// TIA Portal V17 export
// export: Created 2021-09-01T12:00:00, ExportSetting None, DisplayName Totally Integrated Automation Portal, DisplayVersion V17 Update 6
FUNCTION_BLOCK "DEMOSCHRITTKETTE"   // FB45, LAD
TITLE = DemoSchrittKette
{ S7_Optimized_Access := 'TRUE' }
// Auto genereted sequence by graph2LAD: 2024-11-19
// E.R. https://github.com/eliasrhoden
// stored: MemoryReserve 100, SetENOAutomatically false
   VAR_INPUT
      enable : Bool;   // Enables the state machine
      reset : Bool;   // Resets to init state
   END_VAR
   VAR
      statStep : Int;   // Current step/state
      statNextStep : Int;   // Step/State next PLC cycle
   END_VAR
   VAR CONSTANT
      INIT : Int := 0;
      GOTO_HOME : Int := 10;
      AT_HOME_POS : Int := 20;
      LOADING : Int := 30;
      WORKING : Int := 40;
      UNLOADING : Int := 50;
   END_VAR
   VAR_TEMP   // added for the SCL form of the ladder/FBD networks
      _w1 : Bool;
   END_VAR
BEGIN

REGION Network 1 (SCL): Reset
   IF #reset THEN
    #statStep := #INIT;
    #statNextStep := #INIT;
   END_IF;
END_REGION

REGION Network 2: INIT
   // INIT
   // 	 -> GOTO_HOME 
   // 	 -> UNLOADING
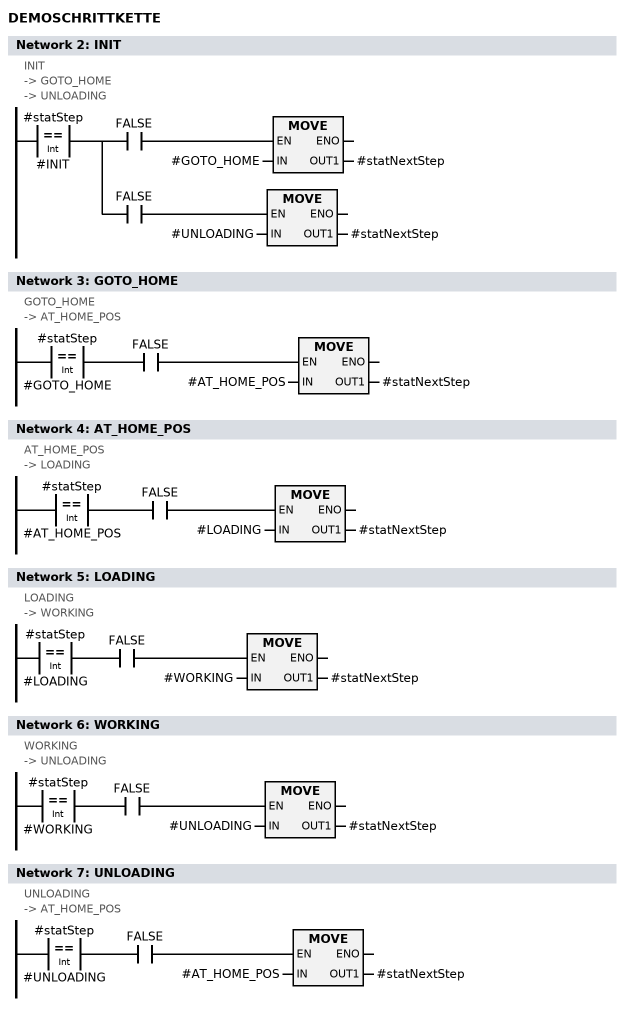
   RUNG wire#powerrail
      { S7_Templates := "SrcType := Int" } EQ_Contact(in1 := #statStep, in2 := #INIT)
      wire#w1
      Contact( FALSE )
      Move(in := #GOTO_HOME, out1 => #statNextStep)
   END_RUNG
   RUNG wire#w1
      Contact( FALSE )
      Move(in := #UNLOADING, out1 => #statNextStep)
   END_RUNG
   // the same network as SCL:
   #_w1 := #statStep = #INIT;
   IF #_w1 AND FALSE THEN
       #statNextStep := #GOTO_HOME;
       #statNextStep := #UNLOADING;
   END_IF;
END_REGION

REGION Network 3: GOTO_HOME
   // GOTO_HOME
   // 	 -> AT_HOME_POS
   RUNG wire#powerrail
      { S7_Templates := "SrcType := Int" } EQ_Contact(in1 := #statStep, in2 := #GOTO_HOME)
      Contact( FALSE )
      Move(in := #AT_HOME_POS, out1 => #statNextStep)
   END_RUNG
   // the same network as SCL:
   IF (#statStep = #GOTO_HOME) AND FALSE THEN #statNextStep := #AT_HOME_POS; END_IF;
END_REGION

REGION Network 4: AT_HOME_POS
   // AT_HOME_POS
   // 	 -> LOADING
   RUNG wire#powerrail
      { S7_Templates := "SrcType := Int" } EQ_Contact(in1 := #statStep, in2 := #AT_HOME_POS)
      Contact( FALSE )
      Move(in := #LOADING, out1 => #statNextStep)
   END_RUNG
   // the same network as SCL:
   IF (#statStep = #AT_HOME_POS) AND FALSE THEN #statNextStep := #LOADING; END_IF;
END_REGION

REGION Network 5: LOADING
   // LOADING
   // 	 -> WORKING
   RUNG wire#powerrail
      { S7_Templates := "SrcType := Int" } EQ_Contact(in1 := #statStep, in2 := #LOADING)
      Contact( FALSE )
      Move(in := #WORKING, out1 => #statNextStep)
   END_RUNG
   // the same network as SCL:
   IF (#statStep = #LOADING) AND FALSE THEN #statNextStep := #WORKING; END_IF;
END_REGION

REGION Network 6: WORKING
   // WORKING
   // 	 -> UNLOADING
   RUNG wire#powerrail
      { S7_Templates := "SrcType := Int" } EQ_Contact(in1 := #statStep, in2 := #WORKING)
      Contact( FALSE )
      Move(in := #UNLOADING, out1 => #statNextStep)
   END_RUNG
   // the same network as SCL:
   IF (#statStep = #WORKING) AND FALSE THEN #statNextStep := #UNLOADING; END_IF;
END_REGION

REGION Network 7: UNLOADING
   // UNLOADING
   // 	 -> AT_HOME_POS
   RUNG wire#powerrail
      { S7_Templates := "SrcType := Int" } EQ_Contact(in1 := #statStep, in2 := #UNLOADING)
      Contact( FALSE )
      Move(in := #AT_HOME_POS, out1 => #statNextStep)
   END_RUNG
   // the same network as SCL:
   IF (#statStep = #UNLOADING) AND FALSE THEN #statNextStep := #AT_HOME_POS; END_IF;
END_REGION

REGION Network 8 (SCL): Next step
   // This ensurers that we remain in each state step at least 1 plc cycle
   IF #enable THEN
    #statStep := #statNextStep;
   END_IF;
END_REGION
END_FUNCTION_BLOCK
